// TIA Portal V18 export
// export: Created 2025-12-01T17:50:36.1573981Z, ExportSetting None, DisplayName Totally Integrated Automation Portal, DisplayVersion V18 Update 5, DisplayName TIA Portal Openness, DisplayVersion V18 Update 5, DisplayName TIA Portal Teamcenter Gateway, DisplayVersion V18, DisplayName TIA Portal Version Control Interface, DisplayVersion V18, DisplayName STEP 7 Professional, DisplayVersion V18 Update 5, DisplayName STEP 7 Safety, DisplayVersion V18, DisplayName WinCC Professional, DisplayVersion V18 Update 5
DATA_BLOCK "TON"   // DB163
{ S7_Optimized_Access := 'TRUE' }
// stored: AutoNumber false, MemoryReserve 100
   VAR
      TON : Array[0..100] of TON_TIME;
      CTU { S7_SetPoint := 'True'} : Array[0..20] of IEC_DCOUNTER;
   END_VAR
   VAR RETAIN
      P { S7_SetPoint := 'True'} : Array[0..20] of Bool;
   END_VAR
BEGIN
END_DATA_BLOCK
